Fanuc TP program (LS listing): MOTN003.LS

/PROG  MOTN003
/ATTR
OWNER		= MNEDITOR;
COMMENT		= "PR_ROB_EZ1/SP1";
PROG_SIZE	= 588;
CREATE		= DATE 10-06-14  TIME 12:00:00;
MODIFIED	= DATE 17-03-27  TIME 17:07:52;
FILE_NAME	= ;
VERSION		= 0;
LINE_COUNT	= 17;
MEMORY_SIZE	= 900;
PROTECT		= READ_WRITE;
TCD:  STACK_SIZE	= 0,
      TASK_PRIORITY	= 50,
      TIME_SLICE	= 0,
      BUSY_LAMP_OFF	= 0,
      ABORT_REQUEST	= 0,
      PAUSE_REQUEST	= 0;
DEFAULT_GROUP	= 1,1,*,*,*;
CONTROL_CODE	= 00000000 00000000;
/MN
    :  !Vorbesetzung Positions-Register ;
    :  !Robotergefuehrte EZ1/SP1 ;
    :  !KS24 ;
    :  !Version: 01 ;
    :  !Stand: 001 ;
    :  !letzte  Aenderung  06.02.2015 LZ ;
    :  UNLOCK PREG ;
    :  PR[11]=LPOS    ;
    :  PR[12]=LPOS    ;
    :  !PR[11] Ruecksetzen ;
    :  CALL PRNULL(11) ;
    :  !PR[12] Ruecksetzen ;
    :  CALL PRNULL(12) ;
    :  !Kappenabnuetzung fester E-Arm EZ ;
    :  PR[GP1:11,1]=(GI[25]*(.1)) ;
    :  !Kappenabnuetzung bewegl. E-Arm E ;
    :  PR[GP2:12,1]=(GI[25]*(-.2)) ;
/POS
/END
